// TIA Portal V15 export
// export: Created 2018-12-10T18:36:36.23961Z, ExportSetting WithDefaults, WithReadOnly, DisplayName Totally Integrated Automation Portal, DisplayVersion V15 Update 2, DisplayName TIA Portal Openness, DisplayVersion V15 Update 2, DisplayName STEP 7 Professional, DisplayVersion V15 Update 2, DisplayName STEP 7 Safety, DisplayVersion V15, DisplayName WinCC Professional, DisplayVersion V15 Update 2, DisplayName SIMATIC Visualization Architect, DisplayVersion V15 Update 1
FUNCTION "VALVENAME_Call" : Void   // FC42, FBD
TITLE = VALVENAME Geo station valve 1 / VALVENAME Geostation Ventil 1
{ S7_Optimized_Access := 'FALSE' }
VERSION : 0.1
// stored: AutoNumber true, CodeModifiedDate 2018-01-29T16:41:45.5621145Z, CompileDate 2018-02-20T10:24:47.6894513Z, CreationDate 2016-05-26T15:39:56.1944252Z, HandleErrorsWithinBlock false, InterfaceModifiedDate 2017-10-27T11:23:28.3952061Z, IsConsistent true, IsIECCheckEnabled false, IsKnowHowProtected false, IsWriteProtected false, LibraryConformanceStatus Error: The block contains calls of single instances. Warning: The object contains access to global data blocks. Warning: The block contains direct access to inputs, outputs, bit memories, indirect access to the registry or indirect access to external memory areas that are unknown at the time of compilation., ModifiedDate 2018-01-29T16:41:45.5621145Z, ParameterModified 2017-10-27T11:23:28.3512036Z, PLCSimAdvancedSupport false, SetENOAutomatically False, StructureModified 2017-10-27T11:23:28.3952061Z, UDAEnableTagReadback false
BEGIN
END_FUNCTION
